// TIA Portal V20 export
DATA_BLOCK "Alarms"   // DB33
{ DB_Accessible_From_OPC_UA := 'FALSE' }
AUTHOR : ERsystem_FA2_DH. Kim
// stored: DBAccessibleFromOPCUA false, DBAccessibleFromWebserver false, MemoryReserve 100, Namespace Unit1.Em7
   VAR
      emAlarms { ExternalWritable := 'False'} : "LAF_typeAlarms";
      maintenanceFaults { ExternalWritable := 'False'} : Array[0..199] of Bool;   // PFE Maintenance Faults
      productionFaults { ExternalWritable := 'False'} : Array[0..199] of Bool;   // PFE Production Faults
      toolingFault { ExternalWritable := 'False'} : Array[0..199] of Bool;   // PFE Tooling Faults
      qualityFault { ExternalWritable := 'False'} : Array[0..199] of Bool;   // PFE Quality Faults
      throughputFaultBlocked { ExternalWritable := 'False'} : Array[0..199] of Bool;   // PFE Throughput Fault Blocked
      throughputFaultStarved { ExternalWritable := 'False'} : Array[0..199] of Bool;   // PFE Throughput Fault Starved
      throughputFault { ExternalWritable := 'False'} : Array[0..199] of Bool;   // PFE Throughput Fault
      systemFaultGeneral { ExternalWritable := 'False'} : Array[0..199] of Bool;   // PFE System Fault General
      materialFault { ExternalWritable := 'False'} : Array[0..199] of Bool;   // PFE Material Fault
      maintenanceWarnings { ExternalWritable := 'False'} : Array[0..199] of Bool;   // PFE Maintenance Warnings
      productionWarning { ExternalWritable := 'False'} : Array[0..199] of Bool;   // PFE Production Warning
      toolingWarning { ExternalWritable := 'False'} : Array[0..199] of Bool;   // PFE Tooling Warning
      qualityWarning { ExternalWritable := 'False'} : Array[0..199] of Bool;   // PFE Quality Warning
      throughputWarning { ExternalWritable := 'False'} : Array[0..199] of Bool;   // PFE Throughput Warning
      systemWarning { ExternalWritable := 'False'} : Array[0..199] of Bool;   // PFE System Warning
      materialWarning { ExternalWritable := 'False'} : Array[0..199] of Bool;   // PFE Material Warning
      maintenanceStatus { ExternalWritable := 'False'} : Array[0..199] of Bool;   // PFE Maintenance Status
      productionStatus { ExternalWritable := 'False'} : Array[0..199] of Bool;   // PFE Production Status
      toolingStatus { ExternalWritable := 'False'} : Array[0..199] of Bool;   // PFE Tooling Status
      qualityStatus { ExternalWritable := 'False'} : Array[0..199] of Bool;   // PFE Quality Status
      throughputStatus { ExternalWritable := 'False'} : Array[0..199] of Bool;   // PFE Throughput Status
      systemStatus { ExternalWritable := 'False'} : Array[0..199] of Bool;   // PFE System Status
      materialStatus { ExternalWritable := 'False'} : Array[0..199] of Bool;   // PFE Material Status
      tonMaintenanceFault { ExternalWritable := 'False'} : Array[0..199] of TON_TIME;   // PFE Maintenance Faults Ton Timer
      tonProductionFault { ExternalWritable := 'False'} : Array[0..199] of TON_TIME;   // PFE Production Faults Ton Timer
      tonToolingFault { ExternalWritable := 'False'} : Array[0..199] of TON_TIME;   // PFE Tooling Faults Ton Timer
      tonQualityFault { ExternalWritable := 'False'} : Array[0..199] of TON_TIME;   // PFE Quality Faults Ton Timer
      tonThroughputFaultBlocked { ExternalWritable := 'False'} : Array[0..199] of TON_TIME;   // PFE Throughput Fault Blocked Ton Timer
      tonThroughputFaultStarved { ExternalWritable := 'False'} : Array[0..199] of TON_TIME;   // PFE Throughput Fault Starved Ton Timer
      tonThroughputFault { ExternalWritable := 'False'} : Array[0..199] of TON_TIME;   // PFE Throughput Fault Ton Timer
      tonSystemFaultGeneral { ExternalWritable := 'False'} : Array[0..199] of TON_TIME;   // PFE System Fault General Ton Timer
      tonMaterialFault { ExternalWritable := 'False'} : Array[0..199] of TON_TIME;   // PFE Material Fault Ton Timer
      tonMaintenanceWarning { ExternalWritable := 'False'} : Array[0..199] of TON_TIME;   // PFE Maintenance Warnings Ton Timer
      tonProductionWarning { ExternalWritable := 'False'} : Array[0..199] of TON_TIME;   // PFE Production Warning Ton Timer
      tonToolingWarning { ExternalWritable := 'False'} : Array[0..199] of TON_TIME;   // PFE Tooling Warning Ton Timer
      tonQualityWarning { ExternalWritable := 'False'} : Array[0..199] of TON_TIME;   // PFE Quality Warning Ton Timer
      tonThroughputWarning { ExternalWritable := 'False'} : Array[0..199] of TON_TIME;   // PFE Throughput Warning Ton Timer
      tonSystemWarning { ExternalWritable := 'False'} : Array[0..199] of TON_TIME;   // PFE System Warning Ton Timer
      tonMaterialWarning { ExternalWritable := 'False'} : Array[0..199] of TON_TIME;   // PFE Material Warning Ton Timer
      tonMaintenanceStatus { ExternalWritable := 'False'} : Array[0..199] of TON_TIME;   // PFE Maintenance Status Ton Timer
      tonProductionStatus { ExternalWritable := 'False'} : Array[0..199] of TON_TIME;   // PFE Production Status Ton Timer
      tonToolingStatus { ExternalWritable := 'False'} : Array[0..199] of TON_TIME;   // PFE Tooling Status Ton Timer
      tonQualityStatus { ExternalWritable := 'False'} : Array[0..199] of TON_TIME;   // PFE Quality Status Ton Timer
      tonThroughputStatus { ExternalWritable := 'False'} : Array[0..199] of TON_TIME;   // PFE Throughput Status Ton Timer
      tonSystemStatus { ExternalWritable := 'False'} : Array[0..199] of TON_TIME;   // PFE System Status Ton Timer
      tonMaterialStatus { ExternalWritable := 'False'} : Array[0..199] of TON_TIME;   // PFE Material Status Ton Timer
      axisErrorCode { ExternalWritable := 'False'} : Array[0..9] of UDInt;
   END_VAR
BEGIN
   emAlarms.error := TRUE;
   emAlarms.warning := FALSE;
   emAlarms.info := FALSE;
   // maintenanceFaults[0] : Sepa Clamp & Cutter safety pin Faults
   // maintenanceFaults[1] : Sepa Gripper safety pin Faults
   // maintenanceFaults[10] : SEPA CLAMP&CUTTER X-AXIS LIMIT SENSOR(-)
   // maintenanceFaults[11] : SEPA CLAMP&CUTTER X-AXIS LIMIT SENSOR(+)
   // maintenanceFaults[12] : SEPA CLAMP&CUTTER Z-AXIS LIMIT SENSOR(-)
   // maintenanceFaults[13] : SEPA CLAMP&CUTTER Z-AXIS LIMIT SENSOR(+)
   // maintenanceFaults[14] : SEPA GRIPPER X-AXIS LIMIT SENSOR(-)
   // maintenanceFaults[15] : SEPA GRIPPER X-AXIS LIMIT SENSOR(+)
   // maintenanceFaults[16] : SEPA GRIPPER Z-AXIS LIMIT SENSOR(-)
   // maintenanceFaults[17] : SEPA GRIPPER Z-AXIS LIMIT SENSOR(+)
   // maintenanceFaults[18] : SEPA GRIPPER C-AXIS LIMIT SENSOR(+)
   // maintenanceFaults[19] : SEPA GRIPPER C-AXIS LIMIT SENSOR(-)
   // maintenanceFaults[20] : JR WINDER FRONT Y-AXIS LIMIT SENSOR(-)
   // maintenanceFaults[21] : JR WINDER FRONT Y-AXIS LIMIT SENSOR(+)
   // maintenanceFaults[22] : JR WINDER REAR Y-AXIS LIMIT SENSOR(-)
   // maintenanceFaults[23] : JR WINDER REAR Y-AXIS LIMIT SENSOR(+)
   // maintenanceFaults[24] : PUSHER ROLLER B-AXIS LIMIT SENSOR(-)
   // maintenanceFaults[25] : PUSHER ROLLER B-AXIS LIMIT SENSOR(+)
   // maintenanceFaults[26] : PUSHER ROLLER Z-AXIS LIMIT SENSOR(-)
   // maintenanceFaults[27] : PUSHER ROLLER Z-AXIS LIMIT SENSOR(+)
   // maintenanceFaults[30] : SEPA CLAMP&CUTTER X-AXIS Drive Fault
   // maintenanceFaults[31] : SEPA CLAMP&CUTTER Z-AXIS Drive Fault
   // maintenanceFaults[32] : SEPA GRIPPER X-AXIS Drive Fault
   // maintenanceFaults[33] : SEPA GRIPPER Z-AXIS Drive Fault
   // maintenanceFaults[34] : SEPA GRIPPER C-AXIS Drive Fault
   // maintenanceFaults[35] : JR WINDER FRONT Y-AXIS Drive Fault
   // maintenanceFaults[36] : JR WINDER REAR Y-AXIS Drive Fault
   // maintenanceFaults[37] : PUSHER ROLLER B-AXIS Drive Fault
   // maintenanceFaults[38] : PUSHER ROLLER Z-AXIS Drive Fault
   // maintenanceFaults[50] : SEPA CLAMP&CUTTER X-AXIS Home Sensor Abnomal
   // maintenanceFaults[51] : SEPA CLAMP&CUTTER Z-AXIS Home Sensor Abnomal
   // maintenanceFaults[52] : SEPA GRIPPER X-AXIS Home Sensor Abnomal
   // maintenanceFaults[53] : SEPA GRIPPER Z-AXIS Home Sensor Abnomal
   // maintenanceFaults[54] : SEPA GRIPPER C-AXIS Home Sensor Abnomal
   // maintenanceFaults[55] : JR WINDER FRONT Y-AXIS Home Sensor Abnomal
   // maintenanceFaults[56] : JR WINDER REAR Y-AXIS Home Sensor Abnomal
   // maintenanceFaults[57] : PUSHER ROLLER B-AXIS Home Sensor Abnomal
   // maintenanceFaults[58] : PUSHER ROLLER Z-AXIS Home Sensor Abnomal
END_DATA_BLOCK
